// TwinCAT 3 PLC project PLC
// ProgramVersion: 3.1.4024.0
// libraries:
//   Tc2_Standard, * (Beckhoff Automation GmbH)
//   Tc2_System, * (Beckhoff Automation GmbH)
//   Tc3_Module, * (Beckhoff Automation GmbH)
//   VisuSymbols,3.5.10.0,System
// project tree:
//   DUTs/ ItemState.TcDUT
//   / GlobalTextList.TcGTLO, PlcTask.TcTTO, Visualization Manager.TcVMO (not stored), Visualization.TcVIS
//   POUs/ MAIN.TcPOU, RobotWorkcenterControl.TcPOU
//   POUs/Simulation/ RobotSimulation.TcPOU, WorkcenterSimulation.TcPOU
// real-time tasks:
//   TASK PlcTask: cycle T#10ms, priority 20, ADS port 350

CONFIGURATION PLC
    RESOURCE PLC ON TwinCAT3
        TASK PlcTask(INTERVAL := T#10ms, PRIORITY := 20);
        PROGRAM MAIN WITH PlcTask : MAIN;
    END_RESOURCE
END_CONFIGURATION

// ---- DUTs/ItemState.TcDUT
TYPE ItemState :
STRUCT
	InProcess	:	BOOL;			// item picked-up by robot & processing by workcenter 
	Done		:	BOOL;			// item processing completed
END_STRUCT
END_TYPE

// ---- POUs/MAIN.TcPOU
PROGRAM MAIN
VAR
	RobotWorkcenterControl			:		RobotWorkcenterControl;
	RobotSimulation					:		RobotSimulation;
	WorkcenterSimulation			:		WorkcenterSimulation;
	
	Start							: 		BOOL;
END_VAR
VAR // added by the converter: edge detectors and wires of the graphical bodies
    _w1 : BOOL;
END_VAR

_w1 := RobotWorkcenterControl.WorkcenterPrgNo > 0;
RobotWorkcenterControl(
    StartProcess := Start,
    RobotPrgDone := RobotSimulation.ProgramDone,
    WorkcenterDone := WorkcenterSimulation.ProgramDone);
RobotSimulation(StartProgramNo := RobotWorkcenterControl.RobotPrgNo, ProgramTime := T#2S);
WorkcenterSimulation(StartProgram := _w1, ProgramTime := T#2S);

END_PROGRAM

// ---- POUs/RobotWorkcenterControl.TcPOU
FUNCTION_BLOCK RobotWorkcenterControl

VAR_INPUT
	StartProcess	:	BOOL;				// machine start
	RobotPrgDone	: 	BOOL;				// input from robot  - program (1 or 2) done
	WorkcenterDone	:	BOOL;				// input from workcenter - program 1 done
END_VAR
VAR_OUTPUT
	InOperation		:	BOOL;				// indication that machine in operation mode
	ReadyForNewTask	:	BOOL;				// indication that machine ready for 25 new items
	
	RobotPrgNo		:	INT:=-1;			// call robot program number
	RobotTakePosX	:	INT;				// pick up position for robot
	RobotTakePosY	:	INT;				// pick up position for robot

	WorkcenterPrgNo	: INT:=-1;				// call workcenter program number (process the item)
END_VAR
VAR CONSTANT
	TableX			:	INT:=5;				// number of items in X direction 
	TableY			:	INT:=5;				// number of items in Y direction
END_VAR
VAR
	ItemsTable		:	ARRAY[1..TableX, 1..TableY] OF ItemState;	// table with items
	RunAll			: 	BOOL;										// run for all items									
	RunOne			: 	BOOL;										// run for one item
END_VAR

IF StartProcess AND ReadyForNewTask THEN
	TableReset();
	ReadyForNewTask := FALSE;			// turn off the task done
	InOperation := TRUE;				// turn on operating mode
	RunAll:=TRUE;
	RunOne:=FALSE;
END_IF

// take next item from the table
IF RunAll AND NOT RunOne THEN
	GetNextItem();
END_IF

// If no more items, then stop
IF RobotTakePosX=0 AND RobotTakePosY=0 THEN
	RunAll:=FALSE;
	ReadyForNewTask:=TRUE;		// operation completed
	InOperation:=FALSE;	// no operating mode
END_IF

// one item is in operating mode
IF RunAll THEN
	Operate();
END_IF

METHOD GetNextItem : BOOL
VAR_INPUT
END_VAR
VAR
	X, Y		: INT;		// index for loop
	Found		: BOOL;		// item is taken
END_VAR
// find the next item to be moved from the table

// reset next item position to zero
RobotTakePosX:=0;
RobotTakePosY:=0;
Found:=FALSE;

// loop all items
// get the last item
FOR X:=1 TO TableX DO
	FOR Y:=1 TO TableY DO
		IF NOT ItemsTable[X,Y].InProcess AND NOT Found THEN
			RobotTakePosX:=X;
			RobotTakePosY:=Y;
			ItemsTable[X,Y].InProcess:=TRUE;	// set as item to pickup
			Found:=TRUE;
		END_IF
	END_FOR
END_FOR
END_METHOD

METHOD Operate : BOOL
VAR_INPUT
END_VAR

VAR

END_VAR
// Send TakeXPos and TakeYPos position to the robot before
// executing the code below

// signal to robot. Move one item
IF NOT RunOne THEN
	RobotPrgNo:=1;			// start robot program 1
END_IF

RunOne:=TRUE;				// one item in progress

// robot task done, start workcenter
IF RobotPrgDone AND RobotPrgNo=1 THEN
	RobotPrgNo:=-1;
	WorkcenterPrgNo:=1;	
END_IF

// workcenter task done, item back to table
IF WorkcenterDone THEN
	WorkcenterPrgNo:=-1;
	RobotPrgNo:=2;
END_IF

// robot task done
IF RobotPrgDone AND RobotPrgNo=2 THEN
	RobotPrgNo:=-1;
	RunOne:=FALSE;			// stop item in progress
	ItemsTable[RobotTakePosX,RobotTakePosY].Done := TRUE;
END_IF
END_METHOD

METHOD TableReset : BOOL
VAR_INPUT
END_VAR
VAR
	X, Y		: INT;		// index for loop
END_VAR
// init new table
// reset all elements in the ARRAY
// set all elements to FALSE i.e. its ready to be moved

FOR X:=1 TO TableX DO
	FOR Y:=1 TO TableY DO
		ItemsTable[X,Y].InProcess := FALSE;
		ItemsTable[X,Y].Done := FALSE;
	END_FOR
END_FOR
END_METHOD

END_FUNCTION_BLOCK

// ---- POUs/Simulation/RobotSimulation.TcPOU
FUNCTION_BLOCK RobotSimulation
VAR_INPUT
	StartProgramNo			:	INT;		// start robot program
	ProgramTime				:	TIME;		// program execution time
END_VAR
VAR_OUTPUT
	ProgramDone				:	BOOL;		// robot program done
	TaskProgress			:	INT;		// completion of current program in percent
	ArmPosition				:	INT;		// arm position for visualisation
END_VAR
VAR
	TimeSim					:	TON;		// robot work timer
END_VAR

TimeSim(IN:=StartProgramNo>0, PT:=ProgramTime, Q=>ProgramDone);

IF ProgramTime<>T#0S THEN
	TaskProgress := 100 * TIME_TO_INT(TimeSim.ET) / TIME_TO_INT(ProgramTime);
END_IF;

IF StartProgramNo < 1 THEN
	ArmPosition:=0;
ELSIF StartProgramNo=1 THEN
	ArmPosition:=(300 + (TaskProgress * 130 / 100)) MOD 360;
ELSIF StartProgramNo=2 THEN
	ArmPosition:=(70 - (TaskProgress * 130 / 100)) MOD 360; 
END_IF

END_FUNCTION_BLOCK

// ---- POUs/Simulation/WorkcenterSimulation.TcPOU
FUNCTION_BLOCK WorkcenterSimulation
VAR_INPUT
	StartProgram			:	BOOL;		// start workcenter program
	ProgramTime				:	TIME;		// program execution time
END_VAR
VAR_OUTPUT
	ProgramDone				:	BOOL;		// workcenter program done
END_VAR
VAR
	TimeSim					:	TON;		// workcenter work timer
END_VAR


TimeSim(IN:=StartProgram, PT:=ProgramTime, Q=>ProgramDone);

END_FUNCTION_BLOCK

// ---- GlobalTextList.TcGTLO
TEXTLIST GlobalTextList
  349 = 'In Operation'
  70 = 'Prg No: %s'
  657 = 'Ready For Task'
  205 = 'Robot'
  390 = 'Start Process'
  241 = 'Workcenter'
END_TEXTLIST

// ---- Visualization.TcVIS
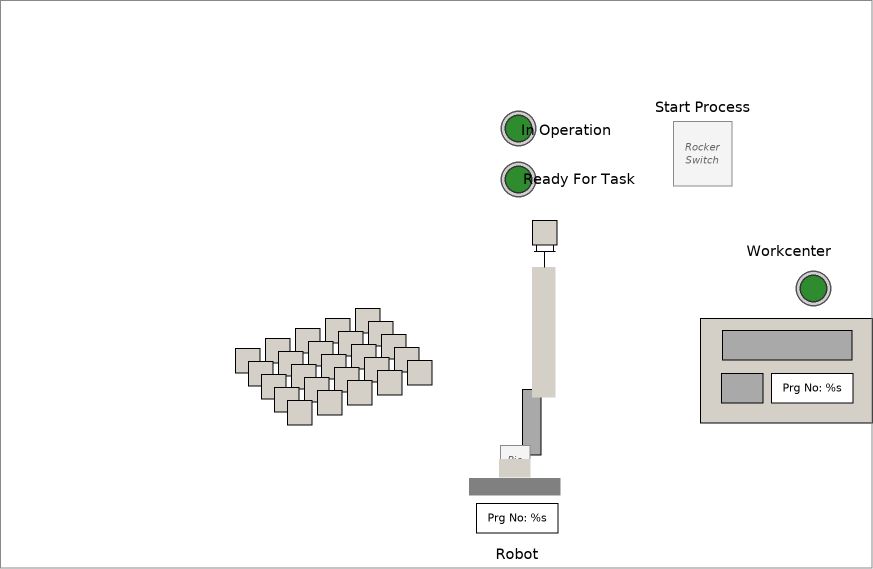
VISUALIZATION Visualization  // 873x569
    RoundedRectangle (522,389 19x66), angle 31, colour toggle: MAIN.RobotWorkcenterControl.RobotPrgNo>0
    RoundedRectangle (355,308 25x25), colour toggle: MAIN.RobotWorkcenterControl.ItemsTable[1,5].Done=TRUE, invisible if: MAIN.RobotWorkcenterControl.ItemsTable[1,5].InProcess=TRUE AND MAIN.RobotWorkcenterControl.ItemsTable[1,5].Done=FALSE
    RoundedRectangle (368,321 25x25), colour toggle: MAIN.RobotWorkcenterControl.ItemsTable[2,5].Done=TRUE, invisible if: MAIN.RobotWorkcenterControl.ItemsTable[2,5].InProcess=TRUE AND MAIN.RobotWorkcenterControl.ItemsTable[2,5].Done=FALSE
    RoundedRectangle (381,334 25x25), colour toggle: MAIN.RobotWorkcenterControl.ItemsTable[3,5].Done=TRUE, invisible if: MAIN.RobotWorkcenterControl.ItemsTable[3,5].InProcess=TRUE AND MAIN.RobotWorkcenterControl.ItemsTable[3,5].Done=FALSE
    RoundedRectangle (394,347 25x25), colour toggle: MAIN.RobotWorkcenterControl.ItemsTable[4,5].Done=TRUE, invisible if: MAIN.RobotWorkcenterControl.ItemsTable[4,5].InProcess=TRUE AND MAIN.RobotWorkcenterControl.ItemsTable[4,5].Done=FALSE
    RoundedRectangle (407,360 25x25), colour toggle: MAIN.RobotWorkcenterControl.ItemsTable[5,5].Done=TRUE, invisible if: MAIN.RobotWorkcenterControl.ItemsTable[5,5].InProcess=TRUE AND MAIN.RobotWorkcenterControl.ItemsTable[5,5].Done=FALSE
    RoundedRectangle (325,318 25x25), colour toggle: MAIN.RobotWorkcenterControl.ItemsTable[1,4].Done=TRUE, invisible if: MAIN.RobotWorkcenterControl.ItemsTable[1,4].InProcess=TRUE AND MAIN.RobotWorkcenterControl.ItemsTable[1,4].Done=FALSE
    RoundedRectangle (338,331 25x25), colour toggle: MAIN.RobotWorkcenterControl.ItemsTable[2,4].Done=TRUE, invisible if: MAIN.RobotWorkcenterControl.ItemsTable[2,4].InProcess=TRUE AND MAIN.RobotWorkcenterControl.ItemsTable[2,4].Done=FALSE
    RoundedRectangle (351,344 25x25), colour toggle: MAIN.RobotWorkcenterControl.ItemsTable[3,4].Done=TRUE, invisible if: MAIN.RobotWorkcenterControl.ItemsTable[3,4].InProcess=TRUE AND MAIN.RobotWorkcenterControl.ItemsTable[3,4].Done=FALSE
    RoundedRectangle (364,357 25x25), colour toggle: MAIN.RobotWorkcenterControl.ItemsTable[4,4].Done=TRUE, invisible if: MAIN.RobotWorkcenterControl.ItemsTable[4,4].InProcess=TRUE AND MAIN.RobotWorkcenterControl.ItemsTable[4,4].Done=FALSE
    RoundedRectangle (377,370 25x25), colour toggle: MAIN.RobotWorkcenterControl.ItemsTable[5,4].Done=TRUE, invisible if: MAIN.RobotWorkcenterControl.ItemsTable[5,4].InProcess=TRUE AND MAIN.RobotWorkcenterControl.ItemsTable[5,4].Done=FALSE
    RoundedRectangle (295,328 25x25), colour toggle: MAIN.RobotWorkcenterControl.ItemsTable[1,3].Done=TRUE, invisible if: MAIN.RobotWorkcenterControl.ItemsTable[1,3].InProcess=TRUE AND MAIN.RobotWorkcenterControl.ItemsTable[1,3].Done=FALSE
    RoundedRectangle (308,341 25x25), colour toggle: MAIN.RobotWorkcenterControl.ItemsTable[2,3].Done=TRUE, invisible if: MAIN.RobotWorkcenterControl.ItemsTable[2,3].InProcess=TRUE AND MAIN.RobotWorkcenterControl.ItemsTable[2,3].Done=FALSE
    RoundedRectangle (321,354 25x25), colour toggle: MAIN.RobotWorkcenterControl.ItemsTable[3,3].Done=TRUE, invisible if: MAIN.RobotWorkcenterControl.ItemsTable[3,3].InProcess=TRUE AND MAIN.RobotWorkcenterControl.ItemsTable[3,3].Done=FALSE
    RoundedRectangle (334,367 25x25), colour toggle: MAIN.RobotWorkcenterControl.ItemsTable[4,3].Done=TRUE, invisible if: MAIN.RobotWorkcenterControl.ItemsTable[4,3].InProcess=TRUE AND MAIN.RobotWorkcenterControl.ItemsTable[4,3].Done=FALSE
    RoundedRectangle (347,380 25x25), colour toggle: MAIN.RobotWorkcenterControl.ItemsTable[5,3].Done=TRUE, invisible if: MAIN.RobotWorkcenterControl.ItemsTable[5,3].InProcess=TRUE AND MAIN.RobotWorkcenterControl.ItemsTable[5,3].Done=FALSE
    RoundedRectangle (265,338 25x25), colour toggle: MAIN.RobotWorkcenterControl.ItemsTable[1,2].Done=TRUE, invisible if: MAIN.RobotWorkcenterControl.ItemsTable[1,2].InProcess=TRUE AND MAIN.RobotWorkcenterControl.ItemsTable[1,2].Done=FALSE
    RoundedRectangle (278,351 25x25), colour toggle: MAIN.RobotWorkcenterControl.ItemsTable[2,2].Done=TRUE, invisible if: MAIN.RobotWorkcenterControl.ItemsTable[2,2].InProcess=TRUE AND MAIN.RobotWorkcenterControl.ItemsTable[2,2].Done=FALSE
    RoundedRectangle (291,364 25x25), colour toggle: MAIN.RobotWorkcenterControl.ItemsTable[3,2].Done=TRUE, invisible if: MAIN.RobotWorkcenterControl.ItemsTable[3,2].InProcess=TRUE AND MAIN.RobotWorkcenterControl.ItemsTable[3,2].Done=FALSE
    RoundedRectangle (304,377 25x25), colour toggle: MAIN.RobotWorkcenterControl.ItemsTable[4,2].Done=TRUE, invisible if: MAIN.RobotWorkcenterControl.ItemsTable[4,2].InProcess=TRUE AND MAIN.RobotWorkcenterControl.ItemsTable[4,2].Done=FALSE
    RoundedRectangle (317,390 25x25), colour toggle: MAIN.RobotWorkcenterControl.ItemsTable[5,2].Done=TRUE, invisible if: MAIN.RobotWorkcenterControl.ItemsTable[5,2].InProcess=TRUE AND MAIN.RobotWorkcenterControl.ItemsTable[5,2].Done=FALSE
    RoundedRectangle (235,348 25x25), colour toggle: MAIN.RobotWorkcenterControl.ItemsTable[1,1].Done=TRUE, invisible if: MAIN.RobotWorkcenterControl.ItemsTable[1,1].InProcess=TRUE AND MAIN.RobotWorkcenterControl.ItemsTable[1,1].Done=FALSE
    RoundedRectangle (248,361 25x25), colour toggle: MAIN.RobotWorkcenterControl.ItemsTable[2,1].Done=TRUE, invisible if: MAIN.RobotWorkcenterControl.ItemsTable[2,1].InProcess=TRUE AND MAIN.RobotWorkcenterControl.ItemsTable[2,1].Done=FALSE
    RoundedRectangle (261,374 25x25), colour toggle: MAIN.RobotWorkcenterControl.ItemsTable[3,1].Done=TRUE, invisible if: MAIN.RobotWorkcenterControl.ItemsTable[3,1].InProcess=TRUE AND MAIN.RobotWorkcenterControl.ItemsTable[3,1].Done=FALSE
    RoundedRectangle (274,387 25x25), colour toggle: MAIN.RobotWorkcenterControl.ItemsTable[4,1].Done=TRUE, invisible if: MAIN.RobotWorkcenterControl.ItemsTable[4,1].InProcess=TRUE AND MAIN.RobotWorkcenterControl.ItemsTable[4,1].Done=FALSE
    RoundedRectangle (287,400 25x25), colour toggle: MAIN.RobotWorkcenterControl.ItemsTable[5,1].Done=TRUE, invisible if: MAIN.RobotWorkcenterControl.ItemsTable[5,1].InProcess=TRUE AND MAIN.RobotWorkcenterControl.ItemsTable[5,1].Done=FALSE
    Lamp1 (478,108 81x41), variable: MAIN.RobotWorkcenterControl.InOperation, style: Lamp-Lamp1-Green
    Lamp1 (772,268 83x41), variable: MAIN.RobotWorkcenterControl.WorkcenterPrgNo > 0, style: Lamp-Lamp1-Green
    Rectangle (700,318 173x105), colour toggle: MAIN.RobotWorkcenterControl.WorkcenterPrgNo > 0
    RoundedRectangle (722,330 130x30), colour toggle: MAIN.RobotWorkcenterControl.WorkcenterPrgNo > 0
    RoundedRectangle (721,373 42x30), colour toggle: MAIN.RobotWorkcenterControl.WorkcenterPrgNo > 0
    RoundedRectangle (771,373 82x30), "Prg No: %s", text variable: MAIN.RobotWorkcenterControl.WorkcenterPrgNo
    RockerSwitch (673,121 59x65), variable: MAIN.Start, behaviour: TOGGLE, style: Switch-RockerSwitch-Gray
    Label (648,92 109x30), "Start Process"
    Label (741,236 96x30), "Workcenter"
    Lamp1 (478,159 81x41), variable: MAIN.RobotWorkcenterControl.ReadyForNewTask, style: Lamp-Lamp1-Green
    Label (518,115 109x30), "In Operation"
    Label (520,164 123x30), "Ready For Task"
    Rectangle (469,478 91x17)
    Pie (500,445 30x30)
    Rectangle (499,459 31x18)
    Rectangle (532,267 23x130), colour toggle: MAIN.RobotWorkcenterControl.RobotPrgNo>0
        p2858320360: MAIN.RobotSimulation.ArmPosition
    RoundedRectangle (476,503 82x30), "Prg No: %s", text variable: MAIN.RobotWorkcenterControl.RobotPrgNo
    Label (469,539 96x30), "Robot"
    Line (544,251) (544,267)
        p2858320360: MAIN.RobotSimulation.ArmPosition
    Line (534,251) (555,251)
        p2858320360: MAIN.RobotSimulation.ArmPosition
    Line (536,233) (536,251)
        p2858320360: MAIN.RobotSimulation.ArmPosition
    Line (553,233) (553,251)
        p2858320360: MAIN.RobotSimulation.ArmPosition
    RoundedRectangle (532,220 25x25), colour toggle: MAIN.RobotWorkcenterControl.RobotPrgNo=2, invisible if: MAIN.RobotWorkcenterControl.RobotPrgNo<=0
        p2858320360: MAIN.RobotSimulation.ArmPosition
END_VISUALIZATION
